FUNCTION F_IssueActuatorCommand : INT
VAR_INPUT
    sDevice       : STRING(50);   // e.g. 'Chariot1', 'Motor3', ...
    bArg          : BOOL;         // see spec: direction or homing flag
    bHasPosition  : BOOL := FALSE;
    nPosition     : DINT := 0;    // used when Motor & !bArg & position present
END_VAR
VAR
    nlen       : INT;
    n         : INT;
    sPrefix   : STRING(50);
    i         : INT;
    sTmp      : STRING(64);
    sIndexStr : STRING(1);
END_VAR

(* ---- basic checks ---- *)
nLen := LEN(sDevice);
IF nLen < 2 THEN
    F_IssueActuatorCommand := -1;
    RETURN;
END_IF;

// last digit "1".."4"
sIndexStr := MID(sDevice, 1, nLen);      // 1 char at position nLen
n := STRING_TO_INT(sIndexStr);

// prefix = everything except last char
sPrefix := LEFT(sDevice, nLen - 1);

(* ---- build "R<n>_" into sTmp ---- *)
sTmp := CONCAT('R', INT_TO_STRING(n));
sTmp := CONCAT(sTmp, '_');

(* ===================== *)
(* Non-motor devices     *)
(* ===================== *)
IF (sPrefix = 'Chariot') OR (sPrefix = 'Compressor') OR (sPrefix = 'Sensor') OR
   (sPrefix = 'HeatExCoupola') OR (sPrefix = 'RegenCoupola') THEN

    sRequestedActuator := CONCAT(sTmp, sPrefix);   // "R<n>_Prefix"

    IF sPrefix = 'Chariot' THEN
        CASE n OF
            1: Tri1_Mot_Cmd.bCommand := bArg;
            2: Tri2_Mot_Cmd.bCommand := bArg;
            3: Tri3_Mot_Cmd.bCommand := bArg;
            4: Tri4_Mot_Cmd.bCommand := bArg;
        END_CASE

    ELSIF sPrefix = 'Compressor' THEN
        CASE n OF
            1: Cmp1_Mot_Cmd.bCommand := bArg;
            3: Cmp2_Mot_Cmd.bCommand := bArg;
            (* n=2,4 handled elsewhere if needed *)
        END_CASE

    ELSIF sPrefix = 'Sensor' THEN
        CASE n OF
            1: Piv1_Mot_Cmd.bCommand := bArg;
        END_CASE

    ELSIF sPrefix = 'HeatExCoupola' THEN
        CASE n OF
            1: Gui1_Mot_Cmd.bCommand := bArg;
        END_CASE

    ELSIF sPrefix = 'RegenCoupola' THEN
        CASE n OF
            3: Gui2_Mot_Cmd.bCommand := bArg;
        END_CASE
    END_IF;

    // <<< return handling for non-motor >>>
    // function returns the global Result:
    //   -1 = failure, 0 = in progress, 1 = success
    F_IssueActuatorCommand := Result;
    RETURN;
END_IF

(* ===================== *)
(* Motor devices         *)
(* ===================== *)
IF sPrefix = 'Motor' THEN
    IF bArg THEN
        (* Homing *)
        sRequestedActuator := CONCAT(sTmp, 'Home');   // "R<n>_Home"
        CASE n OF
            1: Rail1_Mot_Cmd.bHoming := TRUE;
            2: Rail2_Mot_Cmd.bHoming := TRUE;
            3: Rail3_Mot_Cmd.bHoming := TRUE;
            4: Rail4_Mot_Cmd.bHoming := TRUE;
        END_CASE
    ELSE
        (* Normal move *)
        sRequestedActuator := CONCAT(sTmp, 'Motor');  // "R<n>_Motor"
        IF bHasPosition THEN
            CASE n OF
                1: Rail1_Mot_Cmd.nCommand := nPosition;
                2: Rail2_Mot_Cmd.nCommand := nPosition;
                3: Rail3_Mot_Cmd.nCommand := nPosition;
                4: Rail4_Mot_Cmd.nCommand := nPosition;
            END_CASE
        END_IF
    END_IF;

    // <<< return handling for motors >>>
    F_IssueActuatorCommand := Result;
    RETURN;
END_IF

(* Unknown prefix *)
F_IssueActuatorCommand := -3;

END_FUNCTION

(* stored: Version 1.1.0.1, ProductVersion 3.1.4026.11
   POU F_IssueActuatorCommand: Id {039ba84f-c472-4325-8fd5-bb06a032bcc0}, SpecialFunc None *)
